SUBAPPLICATION Uebung_020 (* Subapplication Type *)
  (* Standard: 61499-2 *)
  (* Version 1.0, 2023-10-23, franz *)
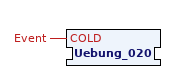
  EVENT_INPUT
    COLD;
  END_EVENT
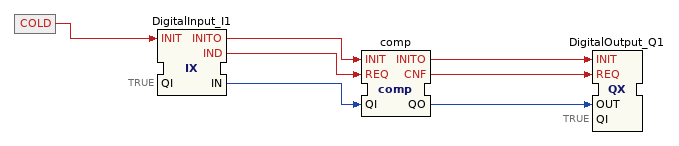
  FBS
    DigitalOutput_Q1 : QX(QI := TRUE);
    DigitalInput_I1 : IX(QI := TRUE);
    comp : comp;
  END_FBS
  EVENT_CONNECTIONS
    COLD TO DigitalInput_I1.INIT;
    DigitalInput_I1.INITO TO comp.INIT;
    comp.INITO TO DigitalOutput_Q1.INIT;
    DigitalInput_I1.IND TO comp.REQ;
    comp.CNF TO DigitalOutput_Q1.REQ;
  END_CONNECTIONS
  DATA_CONNECTIONS
    comp.QO TO DigitalOutput_Q1.OUT;
    DigitalInput_I1.IN TO comp.QI;
  END_CONNECTIONS
END_SUBAPPLICATION
